{attribute 'qualified_only'}
{attribute 'strict'}
TYPE E_ZoneId :
(
    ZONE_NONE       := 0,
    ZONE_A_DRILLING := 1,
    ZONE_B_PROCESS  := 2,
    ZONE_C_LIVING   := 3
);
END_TYPE

(* stored: Version 1.1.0.1, ProductVersion 3.1.4024.16
   DUT E_ZoneId: Id {870f7bdc-dd66-478f-b502-22b03baeef33} *)
